// TIA Portal project "Vinci" (V18)

(* hardware
DEVICE "S7-1200 station_1"  S7-1200 Station
   slot 0: "Rack_0"  S7-1200 Rack  Rack  V1.0
   slot 1: "PLC_1"  CPU 1217C DC/DC/DC  6ES7 217-1AG40-0XB0  V4.6
DEVICE "HMI_1"  TP700 Comfort
   slot 0: "HMI_1"  TP700 Comfort  6AV2 124-0GC01-0AX0  17.0.0.0
   slot 1: "HMI_RT_1"  TP700 Comfort  6AV2 124-0GC01-0AX0  17.0.0.0
   slot 5: "HMI_1.IE_CP_1"  PROFINET Interface  17.0.0.0
      slot 1: "PROFINET Interface_1"  PROFINET Interface
         slot 1: "Port_1"  Port
         slot 2: "Port_2"  Port
   slot 7: "HMI_1.MPI/DP_CP_1"  MPI/DP Interface  17.0.0.0
*)

// ===== PLC "PLC_1"  CPU 1217C DC/DC/DC =====

VAR_GLOBAL   // PLC tag table "IN"
   "Load_Cell_Raw" AT %IW0 : Int;
   "Joystick_Raw" AT %IW2 : Int;
   "Encoder_Raw" AT %ID4 : DInt;
   "Greutate_Incarcatura" AT %ID8 : Real;
   "Buton_Start" AT %I14.0 : Bool;
   "Buton_Stop" AT %I14.1 : Bool;
END_VAR

VAR_GLOBAL   // PLC tag table "OUT"
   "Frana_Mecanica" AT %Q10.0 : Bool;
END_VAR

VAR_GLOBAL   // PLC tag table "MEM"
   "Tensiune_Cablu_kN" AT %MD8 : Real;
   "Joystick_Procent" AT %MD12 : Real;
   "SP_Tensiune_Auto" AT %MD16 : Real;
   "Limita_Warning" AT %M50.0 : Bool;
   "Limita_Trip" AT %M50.1 : Bool;
   "Joystick_Nefiltrat" AT %MD32 : Real;
   "Joystick_Norm" AT %MD36 : Real;
   "Load_Cell_Norm" AT %MD40 : Real;
END_VAR

VAR_GLOBAL   // PLC tag table "BITS"
   "bit1" AT %I12.0 : Bool;
END_VAR

VAR_GLOBAL   // PLC tag table "MOTOR"
   "Viteza_Motor" AT %QD12 : Real;
   "Dir_In" AT %Q20.0 : Bool;
   "Dir_Out" AT %Q20.1 : Bool;
END_VAR

DATA_BLOCK "Joystick_DB"   // DB1
{ S7_Optimized_Access := 'TRUE' }
VERSION : 0.1
// stored: InstanceOfName Joystick
"Joystick"
BEGIN
END_DATA_BLOCK

DATA_BLOCK "Load_Cell_DB"   // DB2
{ S7_Optimized_Access := 'TRUE' }
VERSION : 0.1
// stored: InstanceOfName Load_Cell
"Load_Cell"
BEGIN
END_DATA_BLOCK

DATA_BLOCK "Motor_Control_DB"   // DB3
{ S7_Optimized_Access := 'TRUE' }
VERSION : 0.1
// stored: InstanceOfName Motor_Control
"Motor_Control"
BEGIN
END_DATA_BLOCK

FUNCTION_BLOCK "Joystick"   // FB1, LAD
{ S7_Optimized_Access := 'TRUE' }
VERSION : 0.1
BEGIN

REGION Network 1
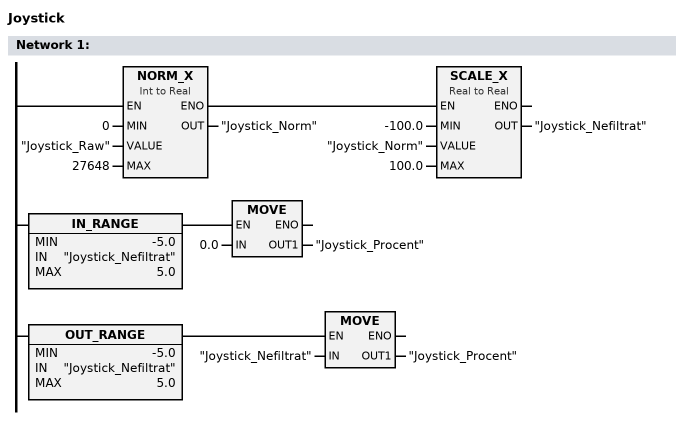
   "Joystick_Norm" := NORM_X(MIN := 0, VALUE := "Joystick_Raw", MAX := 27648);
   "Joystick_Nefiltrat" := SCALE_X(MIN := -100.0, VALUE := "Joystick_Norm", MAX := 100.0);
   IF (-5.0 <= "Joystick_Nefiltrat") AND ("Joystick_Nefiltrat" <= 5.0) THEN
       "Joystick_Procent" := 0.0;
   END_IF;
   IF ("Joystick_Nefiltrat" < -5.0) OR ("Joystick_Nefiltrat" > 5.0) THEN
       "Joystick_Procent" := "Joystick_Nefiltrat";
   END_IF;
END_REGION
END_FUNCTION_BLOCK

FUNCTION_BLOCK "Load_Cell"   // FB2, LAD
{ S7_Optimized_Access := 'TRUE' }
VERSION : 0.1
BEGIN

REGION Network 1
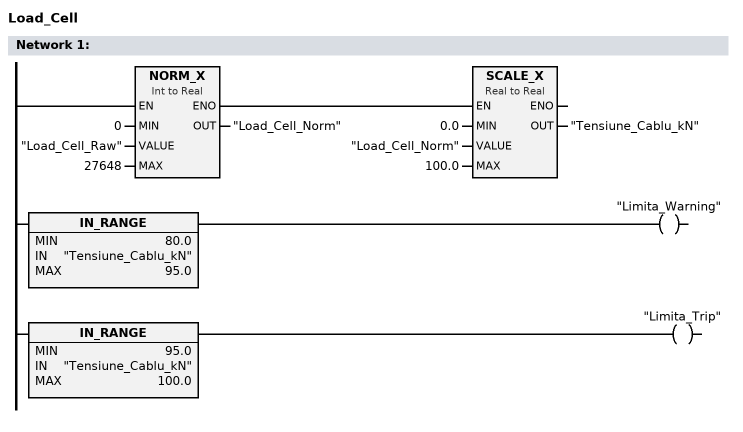
   RUNG wire#powerrail
      { S7_Templates := "[SrcType := Int, DestType := Real]" } Normalize(min := 0, value := "Load_Cell_Raw", max := 27648, out => "Load_Cell_Norm")
      { S7_Templates := "[SrcType := Real, DestType := Real]" } Scale(min := 0.0, value := "Load_Cell_Norm", max := 100.0, out => "Tensiune_Cablu_kN")
   END_RUNG
   RUNG wire#powerrail
      { S7_Templates := "SrcType := Real" } InRange(min := 80.0, in := "Tensiune_Cablu_kN", max := 95.0)
      Coil( "Limita_Warning" )
   END_RUNG
   RUNG wire#powerrail
      { S7_Templates := "SrcType := Real" } InRange(min := 95.0, in := "Tensiune_Cablu_kN", max := 100.0)
      Coil( "Limita_Trip" )
   END_RUNG
   // the same network as SCL:
   "Load_Cell_Norm" := NORM_X(MIN := 0, VALUE := "Load_Cell_Raw", MAX := 27648);
   "Tensiune_Cablu_kN" := SCALE_X(MIN := 0.0, VALUE := "Load_Cell_Norm", MAX := 100.0);
   "Limita_Warning" := (80.0 <= "Tensiune_Cablu_kN") AND ("Tensiune_Cablu_kN" <= 95.0);
   "Limita_Trip" := (95.0 <= "Tensiune_Cablu_kN") AND ("Tensiune_Cablu_kN" <= 100.0);
END_REGION
END_FUNCTION_BLOCK

FUNCTION_BLOCK "Motor_Control"   // FB3, SCL
{ S7_Optimized_Access := 'TRUE' }
VERSION : 0.1
   VAR_INPUT
      in_Joystick_Procent : Real;
      in_Trip_Active : Bool;
      in_Buton_Start : Bool;
      in_Buton_Stop : Bool;
   END_VAR
   VAR_OUTPUT
      out_Cmd_Tragere : Bool;
      out_Cmd_Eliberare : Bool;
      out_Viteza_Ref : Real;
      out_Viteza_Norm : Real;
      out_Viteza_Real : Real;
   END_VAR
   VAR
      stat_Stare_Motor : Bool;
      stat_Viteza_Rampa : Real;
   END_VAR
BEGIN
   IF #in_Buton_Stop OR #in_Trip_Active THEN
       #stat_Stare_Motor := FALSE;
       #out_Viteza_Real := 0.0;
       #stat_Viteza_Rampa := 0.0;
       #out_Cmd_Tragere := FALSE;
       #out_Cmd_Eliberare := FALSE;
   ELSIF #in_Buton_Start THEN
       #stat_Stare_Motor := TRUE;
   END_IF;

   IF #stat_Stare_Motor THEN

       "RampFunction_DB"(
                         Input := #in_Joystick_Procent,
                         SubstituteOutput := 0.0,
                         ErrorAck := FALSE,
                         Reset := NOT #stat_Stare_Motor,
                         Output => #stat_Viteza_Rampa
       );

       IF #stat_Viteza_Rampa > 0.5 THEN
           #out_Cmd_Tragere := TRUE;
           #out_Cmd_Eliberare := FALSE;
       ELSIF #stat_Viteza_Rampa < -0.5 THEN
           #out_Cmd_Tragere := FALSE;
           #out_Cmd_Eliberare := TRUE;
       ELSE
           #out_Cmd_Tragere := FALSE;
           #out_Cmd_Eliberare := FALSE;
       END_IF;

       #out_Viteza_Ref := ABS(#stat_Viteza_Rampa);
       #out_Viteza_Norm := NORM_X(MIN := 0.0, VALUE := #out_Viteza_Ref, MAX := 100.0);
       #out_Viteza_Real := SCALE_X(MIN := 0.0, VALUE := #out_Viteza_Norm, MAX := 120.0);

   ELSE
       #out_Cmd_Tragere := FALSE;
       #out_Cmd_Eliberare := FALSE;
       #out_Viteza_Real := 0.0;
   END_IF;
END_FUNCTION_BLOCK

ORGANIZATION_BLOCK "Main"   // OB1, LAD, ProgramCycle
TITLE = "Main Program Sweep (Cycle)"
{ S7_Optimized_Access := 'TRUE' }
VERSION : 0.1
   VAR_INPUT
      Initial_Call : Bool;   // Initial call of this OB
      Remanence : Bool;   // =True, if remanent data are available
   END_VAR
BEGIN

REGION Network 1
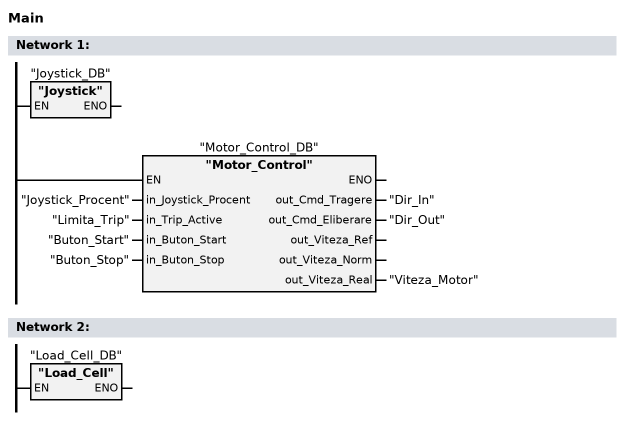
   RUNG wire#powerrail
      "Joystick_DB"()
   END_RUNG
   RUNG wire#powerrail
      "Motor_Control_DB"(in_Joystick_Procent := "Joystick_Procent", in_Trip_Active := "Limita_Trip", in_Buton_Start := "Buton_Start", in_Buton_Stop := "Buton_Stop", out_Cmd_Tragere => "Dir_In", out_Cmd_Eliberare => "Dir_Out", out_Viteza_Ref =>, out_Viteza_Norm =>, out_Viteza_Real => "Viteza_Motor")
   END_RUNG
   // the same network as SCL:
   "Joystick_DB"();   // "Joystick"
   "Motor_Control_DB"(in_Joystick_Procent := "Joystick_Procent",   // "Motor_Control"
                      in_Trip_Active := "Limita_Trip",
                      in_Buton_Start := "Buton_Start",
                      in_Buton_Stop := "Buton_Stop",
                      out_Cmd_Tragere => "Dir_In",
                      out_Cmd_Eliberare => "Dir_Out",
                      out_Viteza_Real => "Viteza_Motor");
END_REGION

REGION Network 2
   RUNG wire#powerrail
      "Load_Cell_DB"()
   END_RUNG
   // the same network as SCL:
   "Load_Cell_DB"();   // "Load_Cell"
END_REGION
END_ORGANIZATION_BLOCK

ORGANIZATION_BLOCK "RampF"   // OB30, SCL, CyclicInterrupt
{ S7_Optimized_Access := 'TRUE' }
VERSION : 0.1
   VAR_INPUT
      Initial_Call : Bool;   // Initial call of this OB
      Event_Count : Int;   // Events discarded
   END_VAR
BEGIN
   "Motor_Control_DB"();
END_ORGANIZATION_BLOCK

(* ===== HMI "HMI_RT_1" =====
system functions are stored by id; their names below are inferred from use
connection "HMI_Connection_1": ETHERNET, S7_1200_OMS

HMI tags "Default tag table"
   "Tag_ScreenNumber" : UInt, internal

HMI tags "IN"
   "Encoder_Raw" : DInt = PLC Encoder_Raw AT %ID4, 1 s
   "Joystick_Raw" : Int = PLC Joystick_Raw AT %IW2, 1 s
   "Load_Cell_Raw" : Int = PLC Load_Cell_Raw AT %IW0, 1 s
   "Greutate_Incarcatura" : Real = PLC Greutate_Incarcatura AT %ID8, 1 s
   "Buton_Start" : Bool = PLC Buton_Start AT %I14.0, 1 s
   "Buton_Stop" : Bool = PLC Buton_Stop AT %I14.1, 1 s

HMI tags "MEM"
   "Tensiune_Cablu_kN" : Real = PLC Tensiune_Cablu_kN AT %MD8, 1 s
   "Joystick_Procent" : Real = PLC Joystick_Procent AT %MD12, 1 s
   "SP_Tensiune_Auto" : Real = PLC SP_Tensiune_Auto AT %MD16, 1 s
   "Limita_Warning" : Bool = PLC Limita_Warning AT %M50.0, 1 s
   "Limita_Trip" : Bool = PLC Limita_Trip AT %M50.1, 1 s
   "Joystick_Nefiltrat" : Real = PLC Joystick_Nefiltrat AT %MD32, 1 s
   "Joystick_Norm" : Real = PLC Joystick_Norm AT %MD36, 1 s
   "Load_Cell_Norm" : Real = PLC Load_Cell_Norm AT %MD40, 1 s

HMI tags "OUT"
   "Frana_Mecanica" : Bool = PLC Frana_Mecanica AT %Q10.0, 1 s

HMI tags "MOTOR"
   "Dir_Out" : Bool = PLC Dir_Out AT %Q20.1, 1 s
   "Dir_In" : Bool = PLC Dir_In AT %Q20.0, 1 s
   "Viteza_Motor" : Real = PLC Viteza_Motor AT %QD12, 1 s

discrete alarms
   1: '', class Errors

screen "Root screen" 800x429, template "Template_1"
   on GenerateScreen: SetTag("Tag_ScreenNumber", 1)
   Button "HmiScreenItemData_1" at 5,363 size 144x56; TextOff 'System screens'; PictureOff "Navigates to System screens for TP1200 Comfort PRO 17.0.0.0"; PictureOn "Navigates to System screens for TP1200 Comfort PRO 17.0.0.0"
      on Release: ActivateScreen("System screens", 0)
   Slider "Slider_1" at 1069,95 size 80x465; Caption 'SIMATIC'
      ProcessValue <- "Joystick_Raw"
   Slider "Slider_2" at 610,36 size 80x383; Caption 'JoyStick'
      ProcessValue <- "Joystick_Raw"
   Circle "Circle_1" at 40,95 size 48x48
      Appearance <- "Limita_Trip"
   Circle "Circle_2" at 40,36 size 48x48
      Appearance <- "Limita_Warning"
   TextField "Text field_1" at 5,12 size 147x23; Text 'Load Warning'
   TextField "Text field_2" at 23,145 size 108x23; Text 'Load Trip'
   TextField "Text field_5" at 439,109 size 16x23; Text 'Text'
   Button "Button_1" at 332,387 size 62x32; TextOff 'Start'
      on Press: SetBit("Buton_Start"); ResetBit("Buton_Stop")
   Button "Button_2" at 408,387 size 62x32; TextOff 'Stop'
      on Press: SetBit("Buton_Stop"); ResetBit("Buton_Start")
   Circle "Circle_3" at 464,5 size 48x48
      Appearance <- "Buton_Start"
   TextField "Text field_9" at 446,50 size 93x24; Text 'Running'
      Appearance <- "Buton_Start"
   TextField "Text field_4" at 315,74 size 54x62; Text '◄'
      Appearance <- "Dir_Out"
   TextField "Text field_3" at 485,74 size 54x62; Text '►'
      Appearance <- "Dir_In"
   IOField "I/O field_1" at 314,131 size 233x37; FormatPattern 999
      ProcessValue <- "Viteza_Motor"
   TextField "Text field_6" at 379,88 size 95x38; Text 'Speed'
   TextField "Text field_7" at 314,13 size 114x25; Text 'Info View'
   TextField "Text field_8" at 455,134 size 70x31; Text 'mpm'

Template "Template_1" 800x429
   Button "Exit" at 1200,679 size 78x59; TextOff 'Exit'; PictureOff "ExitRuntime_TP1200_Comfort_PRO_TR"; PictureOn "ExitRuntime_TP1200_Comfort_PRO_TR"
      on Release: StopRuntime(0)
   Button "Log on" at 1120,679 size 78x59; TextOff 'Log on'; PictureOff "Login_TP1200_Comfort_PRO_TR"; PictureOn "Login_TP1200_Comfort_PRO_TR"
      on Release: function_a2a04561()
   Button "Template_Button" at 1040,679 size 78x59; TextOff 'Text'
   Button "Template_Button_1" at 960,679 size 78x59; TextOff 'Text'
   Button "Template_Button_2" at 880,679 size 78x59; TextOff 'Text'
   Button "Template_Button_3" at 800,679 size 78x59; TextOff 'Text'
   Button "Template_Button_4" at 720,679 size 78x59; TextOff 'Text'
   Button "Template_Button_5" at 640,679 size 78x59; TextOff 'Text'
   Button "Template_Button_6" at 561,679 size 78x59; TextOff 'Text'
   Button "Template_Button_7" at 481,679 size 78x59; TextOff 'Text'
   Button "Template_Button_8" at 401,679 size 78x59; TextOff 'Text'
   Button "Template_Button_9" at 321,679 size 78x59; TextOff 'Text'
   Button "Template_Button_10" at 241,679 size 78x59; TextOff 'Text'
   Button "Language" at 161,679 size 78x59; TextOff 'Language'; PictureOff "ToggleLanguage_TP1200_Comfort_PRO_TR"; PictureOn "ToggleLanguage_TP1200_Comfort_PRO_TR"
      on Release: function_fb9197e8(-1)
   Button "Start screen" at 81,679 size 78x59; TextOff 'Start screen'; PictureOff "NavigateHome_TP1200_Comfort_PRO_TR"; PictureOn "NavigateHome_TP1200_Comfort_PRO_TR"
      on Release: ActivateScreen("Root screen", 0)
   Button "Alarms" at 1,679 size 78x59; TextOff 'Alarms'; PictureOff "AlarmDisplay_TP1200_Comfort_PRO_TR"; PictureOn "AlarmDisplay_TP1200_Comfort_PRO_TR"
      on Release: function_ef3f5d25("Alarm window_Unacknowledged", -1)

screen "System screens" 800x429, template "Template_1"
   on GenerateScreen: SetTag("Tag_ScreenNumber", 2)
   Button "Back" at 1,1 size 159x47; TextOff 'Back'
      on Release: ActivateScreen("Root screen", 0)
   Button "HmiScreenItemData" at 36,95 size 159x47; TextOff 'SIMATIC PLC system diagnos...'; PictureOff "Navigates to SIMATIC PLC system diagnostics for TP1200 Comfort PRO 17.0.0.0"; PictureOn "Navigates to SIMATIC PLC system diagnostics for TP1200 Comfort PRO 17.0.0.0"
      on Release: ActivateScreen("SIMATIC PLC system diagnostics", 0)
   Button "HmiScreenItemData_1" at 36,154 size 159x47; TextOff 'System settings'; PictureOff "Navigates to System settings for TP1200 Comfort PRO 17.0.0.0"; PictureOn "Navigates to System settings for TP1200 Comfort PRO 17.0.0.0"
      on Release: ActivateScreen("System settings", 0)
   Button "HmiScreenItemData_2" at 36,213 size 159x47; TextOff 'System information'; PictureOff "Navigates to System information for TP1200 Comfort PRO 17.0.0.0"; PictureOn "Navigates to System information for TP1200 Comfort PRO 17.0.0.0"
      on Release: ActivateScreen("System information", 0)

screen "SIMATIC PLC system diagnostics" 800x429, template "Template_1"
   on GenerateScreen: SetTag("Tag_ScreenNumber", 3)
   SysDiagControl "HmiScreenItemData" at 1,49 size 1276x623
   Button "Back" at 1,1 size 159x47; TextOff 'Back'
      on Release: ActivateScreen("System screens", 0)

screen "System settings" 800x429, template "Template_1"
   on GenerateScreen: SetTag("Tag_ScreenNumber", 4)
   Button "Clean screen" at 36,95 size 159x47; TextOff 'Clean screen'
      on Release: function_be740847(30)
   Button "Back" at 1,1 size 159x47; TextOff 'Back'
      on Release: ActivateScreen("System screens", 0)

screen "System information" 800x429, template "Template_1"
   on GenerateScreen: SetTag("Tag_ScreenNumber", 5)
   TextField "HmiScreenItemData" at 35,51 size 171x28; Text 'HMI device type:'
   TextField "HmiScreenItemData_1" at 241,51 size 1004x28; Text 'TP1200 Comfort PRO 17.0.0.0'
   TextField "HmiScreenItemData_2" at 35,81 size 171x28; Text 'Version:'
   TextField "HmiScreenItemData_3" at 35,111 size 171x28; Text 'Connection:'
   TextField "HmiScreenItemData_4" at 241,111 size 1004x28; Text 'ETHERNET'
   TextField "HmiScreenItemData_5" at 35,141 size 171x28; Text 'PLC:'
   TextField "HmiScreenItemData_6" at 241,141 size 1004x28; Text 'SIMATIC S7 1200'
   Button "Display version" at 241,81 size 1004x28; TextOff 'Display version'
      on Release: function_febcb963(-1)
   Button "Back" at 1,1 size 159x47; TextOff 'Back'
      on Release: ActivateScreen("System screens", 0)
*)